// TIA Portal V20 export
TYPE "LER_typeSoftCam"
// stored: Access Published
   STRUCT
      Pos0 { S7_SetPoint := 'True'} : "LER_typeSoftCamPosition";
      Pos1 { S7_SetPoint := 'True'} : "LER_typeSoftCamPosition";
      Pos2 { S7_SetPoint := 'True'} : "LER_typeSoftCamPosition";
      Pos3 { S7_SetPoint := 'True'} : "LER_typeSoftCamPosition";
      Pos4 { S7_SetPoint := 'True'} : "LER_typeSoftCamPosition";
      Pos5 { S7_SetPoint := 'True'} : "LER_typeSoftCamPosition";
      Pos6 { S7_SetPoint := 'True'} : "LER_typeSoftCamPosition";
      Pos7 { S7_SetPoint := 'True'} : "LER_typeSoftCamPosition";
      Pos8 { S7_SetPoint := 'True'} : "LER_typeSoftCamPosition";
      Pos9 { S7_SetPoint := 'True'} : "LER_typeSoftCamPosition";
      Pos10 { S7_SetPoint := 'True'} : "LER_typeSoftCamPosition";
      Pos11 { S7_SetPoint := 'True'} : "LER_typeSoftCamPosition";
      Pos12 { S7_SetPoint := 'True'} : "LER_typeSoftCamPosition";
      Pos13 { S7_SetPoint := 'True'} : "LER_typeSoftCamPosition";
      Pos14 { S7_SetPoint := 'True'} : "LER_typeSoftCamPosition";
      Pos15 { S7_SetPoint := 'True'} : "LER_typeSoftCamPosition";
   END_STRUCT;
END_TYPE
